(* PLC project  *)
(* stored: company Example Corp, product Fault Diagnosis, version 1.0 *)

FUNCTION_BLOCK FaultDiagnosis
  VAR_INPUT
    Input1 : REAL;
  END_VAR
  VAR_OUTPUT
    Output1 : REAL;
  END_VAR

(* FBD diagram, written out as Structured Text *)
END_FUNCTION_BLOCK
